FUNCTION_BLOCK XSLIDE_CTL (* Transfer Slide/Clamp Sequence *)
  (* Standard: 61499-1; Classification: Simulation; ApplicationDomain: Machining; Function: Transfer Slide *)
  (* Version 0.0, 2002-10-04, JHC, Rockwell Automation, Modified from DRILL_CTL *)
  (* Compiler header: package fb.rt.mach; *)
  (* Compiler Java IBM Jikes 1.06 *)
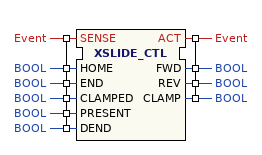
  EVENT_INPUT
    SENSE WITH HOME, END, CLAMPED, PRESENT, DEND; (* Slide+Machine Sensors *)
  END_EVENT
  EVENT_OUTPUT
    ACT WITH FWD, REV, CLAMP; (* Slide actuators *)
  END_EVENT
  VAR_INPUT
    HOME : BOOL; (* Slide at HOME position *)
    END : BOOL; (* Slide at END position *)
    CLAMPED : BOOL; (* Clamp at END position *)
    PRESENT : BOOL; (* Workpiece present on Slide *)
    DEND : BOOL; (* Tool at END position *)
  END_VAR
  VAR_OUTPUT
    FWD : BOOL; (* Advance slide *)
    REV : BOOL; (* Retract slide *)
    CLAMP : BOOL; (* Clamp command, 0=open, 1=close *)
  END_VAR
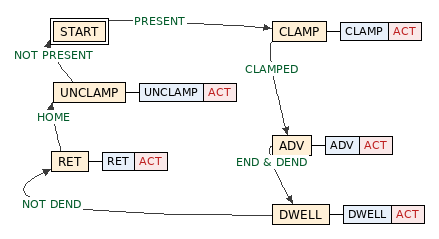
  EC_STATES
    START; (* Initial State *)
    CLAMP : CLAMP -> ACT; (* Clamp Workpiece *)
    ADV : ADV -> ACT; (* Advance Slide *)
    DWELL : DWELL -> ACT; (* Tool Dwell Period *)
    RET : RET -> ACT; (* Return Slide *)
    UNCLAMP : UNCLAMP -> ACT; (* Unclamp Workpiece *)
  END_STATES
  EC_TRANSITIONS
    START TO CLAMP := PRESENT;
    CLAMP TO ADV := CLAMPED;
    ADV TO DWELL := END & DEND;
    DWELL TO RET := NOT DEND;
    RET TO UNCLAMP := HOME;
    UNCLAMP TO START := NOT PRESENT;
  END_TRANSITIONS
  ALGORITHM DWELL IN ST: (* Turn off FWD while machining *)
FWD := false;
  END_ALGORITHM
  ALGORITHM CLAMP IN ST: (* Clamp Workpiece *)
CLAMP := true;
  END_ALGORITHM
  ALGORITHM ADV IN ST: (* Advance Slide *)
FWD:=true;
REV:=false;
  END_ALGORITHM
  ALGORITHM RET IN ST: (* Retract Slide *)
FWD:= false;
REV := true;
  END_ALGORITHM
  ALGORITHM UNCLAMP IN ST: (* Unclamp Workpiece *)
CLAMP := false;
REV := false;
  END_ALGORITHM
END_FUNCTION_BLOCK
